TYPE Structure_RobotPose :
STRUCT
	xPose : INT;
	yPose : INT;
	zPose : INT;
	oPose : INT;
	aPose : INT;
	tPose : INT;
END_STRUCT
END_TYPE

(* stored: Version 1.1.0.1, ProductVersion 3.1.4024.12
   DUT Structure_RobotPose: Id {e2223736-10fa-4632-bd16-3b0278ad8845} *)
